// TwinCAT 3 PLC project CamTest
// ProgramVersion: 3.1.4024.0
// libraries:
//   Tc2_MC2, * (Beckhoff Automation GmbH)
//   Tc2_MC2_Camming, * (Beckhoff Automation GmbH)
//   Tc2_Standard, * (Beckhoff Automation GmbH)
//   Tc2_System, * (Beckhoff Automation GmbH)
//   Tc3_Module, * (Beckhoff Automation GmbH)
// project tree:
//   / PlcTask.TcTTO
//   POUs/ MAIN.TcPOU
// real-time tasks:
//   TASK PlcTask: cycle T#10ms, priority 20, ADS port 350

CONFIGURATION CamTest
    RESOURCE PLC ON TwinCAT3
        TASK PlcTask(INTERVAL := T#10ms, PRIORITY := 20);
        PROGRAM MAIN WITH PlcTask : MAIN;
    END_RESOURCE
END_CONFIGURATION

// ---- POUs/MAIN.TcPOU
PROGRAM MAIN
VAR
	axis1 : AXIS_REF;
	axis2 : AXIS_REF;
	
	axis3 : AXIS_REF;
	axis4 : AXIS_REF;
	
	mcpower1 : MC_Power;
	mcpower2 : MC_Power;
	
	mcpower3 : MC_Power;
	mcpower4 : MC_Power;
	
	mcgearin : MC_GearIn;
	mcMoveAbsoluteAxis3 : MC_MoveAbsolute;
	iGearStep : INT;
	poweron2 : BOOL;
	
	mccamin : MC_CamIn;
	mccamout : MC_CamOut;
	
	allow : BOOL;
	poweron : BOOL;
	
	
	
	
	bAllowGearin: BOOL;
END_VAR

axis1.ReadStatus();
axis2.ReadStatus();
axis3.ReadStatus();
axis4.ReadStatus();
Act();
pCam();
pGear();

ACTION ACT:
mcpower1(
	Axis:=axis1 , 
	Enable:=poweron , 
	Enable_Positive:=poweron , 
	Enable_Negative:=poweron , 
	Override:= , 
	BufferMode:= , 
	Options:= , 
	Status=> , 
	Busy=> , 
	Active=> , 
	Error=> , 
	ErrorID=> );
	
	mcpower2(
	Axis:=axis2 , 
	Enable:=poweron , 
	Enable_Positive:=poweron , 
	Enable_Negative:=poweron , 
	Override:= , 
	BufferMode:= , 
	Options:= , 
	Status=> , 
	Busy=> , 
	Active=> , 
	Error=> , 
	ErrorID=> );
		
    mcpower3(
	Axis:=axis3 , 
	Enable:=poweron2 , 
	Enable_Positive:=poweron2 , 
	Enable_Negative:=poweron2 , 
	Override:= , 
	BufferMode:= , 
	Options:= , 
	Status=> , 
	Busy=> , 
	Active=> , 
	Error=> , 
	ErrorID=> );
		
    mcpower4(
	Axis:=axis4 , 
	Enable:=poweron2 , 
	Enable_Positive:=poweron2 , 
	Enable_Negative:=poweron2 , 
	Override:= , 
	BufferMode:= , 
	Options:= , 
	Status=> , 
	Busy=> , 
	Active=> , 
	Error=> , 
	ErrorID=> );
	
	mcgearin(
	Master:=axis3 , 
	Slave:=axis4 , 
	Execute:= , 
	RatioNumerator:=1 , 
	RatioDenominator:=1 , 
	Acceleration:= , 
	Deceleration:= , 
	Jerk:= , 
	BufferMode:= , 
	Options:= , 
	InGear=> , 
	Busy=> , 
	Active=> , 
	CommandAborted=> , 
	Error=> , 
	ErrorID=> );
	
    mcMoveAbsoluteAxis3(
	Axis:=axis3 , 
	Execute:= , 
	Position:= , 
	Velocity:= , 
	Acceleration:= , 
	Deceleration:= , 
	Jerk:= , 
	BufferMode:= , 
	Options:= , 
	Done=> , 
	Busy=> , 
	Active=> , 
	CommandAborted=> , 
	Error=> , 
	ErrorID=> );
	
	mccamin(
	Master:=axis1 , 
	Slave:=axis2 , 
	Execute:= , 
	MasterOffset:= , 
	SlaveOffset:= , 
	MasterScaling:= , 
	SlaveScaling:= , 
	StartMode:= , 
	CamTableID:=1 , 
	BufferMode:= , 
	Options:= , 
	InSync=> , 
	Busy=> , 
	Active=> , 
	CommandAborted=> , 
	Error=> , 
	ErrorID=> );
END_ACTION

ACTION pCam:
mccamin.Options.ActivationMode := MC_CAMACTIVATION_INSTANTANEOUS;

IF allow THEN
	mccamin.Execute := TRUE;
END_IF
END_ACTION

ACTION pGear:
CASE iGearStep OF
	0:
    IF poweron2 THEN
		iGearStep := 1;
    END_IF
    1:
	IF axis3.Status.ControlLoopClosed AND axis4.Status.ControlLoopClosed THEN
		iGearStep := 2;
	END_IF
    2:
    IF bAllowGearin THEN
		iGearStep := 3;
    END_IF
    3:
	mcgearin.Execute := TRUE;
    mcMoveAbsoluteAxis3.Execute := TRUE;
    mcMoveAbsoluteAxis3.Position := 20;
	mcMoveAbsoluteAxis3.Velocity := 0.4;
    IF mcMoveAbsoluteAxis3.Done THEN
		mcMoveAbsoluteAxis3.Execute := FALSE;
		iGearStep := 4;
	END_IF
    4:
	mcMoveAbsoluteAxis3.Execute := TRUE;
	mcMoveAbsoluteAxis3.Position := 0;
	mcMoveAbsoluteAxis3.Velocity := 0.4;
	IF mcMoveAbsoluteAxis3.Done THEN
		mcMoveAbsoluteAxis3.Execute := FALSE;
		iGearStep :=2;
	END_IF
	
END_CASE
END_ACTION

END_PROGRAM
